{attribute 'linkalways'} 
{attribute 'no_explicit_call' := 'This FB is a CLASS and must be accessed using methods or properties'}
{attribute 'enable_dynamic_creation'}
FUNCTION_BLOCK Node_F_VN_ContourInertiaRatio EXTENDS VisionNode
VAR
    ipContour : _ITcVnContainer;
    fInertiaRatio : _LREAL(0.0);
    hrPrev : _HRESULT(S_OK);
	hresult : _HRESULT(S_OK);
END_VAR

METHOD PUBLIC  Clone : I_Node
VAR
	pNode : POINTER TO Node_F_VN_ContourInertiaRatio;
END_VAR
pNode := __NEW(Node_F_VN_ContourInertiaRatio);
Clone := pNode^;
END_METHOD

METHOD FB_init : BOOL
VAR_INPUT
	bInitRetains : BOOL; // if TRUE, the retain variables are initialized (warm start / cold start)
	bInCopyCode : BOOL;  // if TRUE, the instance afterwards gets moved into the copy code (online change)
END_VAR
AddInput('ipContour', ipContour);
AddInput('hrPrev', hrPrev);
AddOutput('fInertiaRatio', fInertiaRatio);
AddOutput('hresult',hresult);
END_METHOD

METHOD PROTECTED OnExecute
hresult.Value := F_VN_ContourInertiaRatio(
	ipContour := ipContour.Value,
    fInertiaRatio := fInertiaRatio.Value,
	hrPrev:= hrPrev.Value);
END_METHOD

METHOD PUBLIC PreExecutionCheck
VAR_INPUT
	Check : I_PreExecutionChecks;
END_VAR
Check.IsTrue(ipContour.IsValid, 'ipContour must be a valid container');
Check.IsTrue((ipContour.IsType(TC_GLOBAL_CONST_LIST.ContainerType_Vector_TcVnPoint2_DINT) OR
              ipContour.IsType(TC_GLOBAL_CONST_LIST.ContainerType_Vector_TcVnPoint2_REAL)),
              'ipContour contains incorrect type');
END_METHOD

END_FUNCTION_BLOCK

(* stored: Version 1.1.0.1, ProductVersion 3.1.4026.13
   POU Node_F_VN_ContourInertiaRatio: Id {ed47f679-c379-0cbd-356e-36f296f64a5e}, SpecialFunc None
   Folder Constructor: Id {2e91d4de-1ffe-01ed-3bed-2aa7f6088a2b}
   Method Clone: Id {1375420b-fe27-0af8-118f-f650e6394b52}
   Method FB_init: Id {f5e54fab-0c9d-08b5-38e6-01001473a406}
   Method OnExecute: Id {a26a4796-ead7-0ed4-01a8-de94bb244b56}
   Method PreExecutionCheck: Id {0d20fe15-8fa9-026d-0319-f4619437e0bc} *)
